{attribute 'GeneratedUsingTerminal: BK1120-0000-0001'}
{attribute addProperty BoxType "BK1120-0000-0001"}
{attribute addProperty Id "InputsAT %I*Inputs_CC16D1F40OutputsAT %I*Outputs_D8BAB3B30WcStateAT %I*WcState_9091E0EB2InfoDataAT %I*InfoData_41C547A32"}
{attribute addProperty CRC "323002079"}
{attribute addProperty Size "4"}
TYPE BK1120_13409EDF EXTENDS EtcSlaveTerminalBase_947E5A46 :
STRUCT
	{attribute addProperty Name "Inputs"}
	Inputs : Inputs_CC16D1F4;
	{attribute addProperty Name "Outputs"}
	Outputs : Outputs_D8BAB3B3;
	{attribute addProperty Name "WcState"}
	WcState : WcState_9091E0EB;
	{attribute addProperty Name "InfoData"}
	InfoData : InfoData_41C547A3;
END_STRUCT
END_TYPE

(* stored: Version 1.2.0.0, ProductVersion 3.1.4024.9
   DUT BK1120_13409EDF: Id {ed72db71-2a6f-478b-b5fa-f49471dd4607} *)
